ABB RobotStudio station: P2_Main_2.rspag

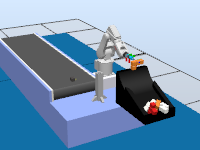
--- station ---
Station P2_Main (saved by RobotStudio 21.1.9385.0)
Controller Controller2, task T_ROB1: task frame (RAPID world) sits at (1547.5, 1227.5, 510) mm in the station
Controller Controller2
  mechanical unit ROB_1: IRB120_3_58__01, 6 joints, base frame (0, 0, 0) mm
Layout (positions relative to the parent item):
  - IRB120_3_58__01 [mechanism, from Robots\IRB120_3_58_G_01.rslib] at (1547.5, 1227.5, 510) mm; joint values [0.0586, 0.4229, 0.2961, 0.0888, -0.7209, -0.0668] (rad or m)
  - MyNewTool [mechanism] at (2003, 1250, 900) mm, rotated rx 0 ry 90 rz 0 deg
      TCP MyNewTool at (0, 0, 0) mm, rotated rx 180 ry 0 rz 180 deg
      links: Čep
  - smc_gripper [mechanism, from Parts\smc_gripper.rslib] at (2003, 1250, 900) mm, rotated rx 0 ry 90 rz 0 deg
  - Conv_belt [part] at (-460, 1030, 390) mm, rotated rx 90 ry 0 rz 0 deg
  - Piece_6_L [part] at (2225, 1200, 885.87) mm, rotated rx 0.75 ry 90 rz 90.75 deg
  - Piece_5_S [part] at (2593.69, 1136.23, 500.91) mm, rotated rx -150.15 ry -50.3 rz 82.94 deg
  - Piece_4_T [part] at (2653.03, 1162.05, 521.4) mm, rotated rx -177.09 ry 74.17 rz -180 deg
  - Piece_2_S [part] at (2730.75, 1281.49, 507.1) mm, rotated rx 90 ry 0 rz -176.34 deg
  - Piece_3_L [part] at (2613.74, 1242.05, 481.96) mm, rotated rx -48.71 ry -65.02 rz -0.13 deg
  - Piece_1_T [part] at (3053.29, 1610.48, 33) mm, rotated rx -95.26 ry 5.23 rz -57.48 deg
  - FLIP [part] at (1915, 935, 785) mm, rotated rx 180 ry 0 rz 90 deg
  - PICKUP [part] at (1493.35, 765, 526.5) mm, rotated rx -90 ry 0 rz -90 deg
  - FlipperStand [part] at (1945, 900, 360) mm, rotated rx 90 ry 0 rz 0 deg
  - Environment_6 [part]
  - DROP [part] at (2100, 1525, 950) mm, rotated rx 0 ry 90 rz -90 deg
  - Positioner_1 [smart component, from Components\Positioner.rslib] at (495, 765, 531.5) mm, rotated rx -90 ry 0 rz 0 deg
      properties: Object=Piece_1_T; Position=[0.5 0.765 0.5315]; Orientation=[-1.5707963267949 0 -1.5707963267949]; Reference=Global; ReferenceObject=(none)
  - Positioner_2 [smart component, from Components\Positioner.rslib] at (2954.8, 1487.14, 42.26) mm, rotated rx -84.7 ry -5.18 rz 122.52 deg
      properties: Object=Piece_2_S; Position=[0.35 0.715 0.5315]; Orientation=[-1.5707963267949 0 1.5707963267949]; Reference=Global; ReferenceObject=(none)
  - Positioner_3 [smart component, from Components\Positioner.rslib] at (2714.8, 1530.98, 507.18) mm, rotated rx 89.95 ry 0.02 rz -86.34 deg
      properties: Object=Piece_3_L; Position=[0.1 0.715 0.5315]; Orientation=[-1.5707963267949 0 0]; Reference=Global; ReferenceObject=(none)
  - Positioner_4 [smart component, from Components\Positioner.rslib] at (2552.24, 1285.06, 88.21) mm, rotated rx -95.3 ry 5.18 rz -57.48 deg
      properties: Object=Piece_4_T; Position=[-0.1 0.765 0.5315]; Orientation=[-1.5707963267949 0 -1.5707963267949]; Reference=Global; ReferenceObject=Piece_4_T
  - Positioner_5 [smart component, from Components\Positioner.rslib] at (-250, 715, 531.5) mm, rotated rx -90 ry 0 rz 90 deg
      properties: Object=Piece_5_S; Position=[-0.25 0.715 0.5315]; Orientation=[-1.5707963267949 0 1.5707963267949]; Reference=Global; ReferenceObject=(none)
  - Positioner_6 [smart component, from Components\Positioner.rslib] at (2676.51, 2129.75, 507.42) mm, rotated rx 89.95 ry 0.02 rz -86.34 deg
      properties: Object=Piece_6_L; Position=[-0.5 0.715 0.5315]; Orientation=[-1.5707963267949 0 0]; Reference=Global; ReferenceObject=(none)
  - Attacher_1_G [smart component, from Components\Attacher.rslib]
      properties: Parent=smc_gripper; Flange=0; Child=Piece_1_T; Mount=false; Offset=[0 0 0]; Orientation=[0 0 0]
  - Attacher_2_G [smart component, from Components\Attacher.rslib]
      properties: Parent=smc_gripper; Flange=0; Child=Piece_2_S; Mount=false; Offset=[0 0 0]; Orientation=[0 0 0]
  - Attacher_3_G [smart component, from Components\Attacher.rslib]
      properties: Parent=smc_gripper; Flange=0; Child=Piece_3_L; Mount=false; Offset=[0 0 0]; Orientation=[0 0 0]
  - Attacher_4_G [smart component, from Components\Attacher.rslib]
      properties: Parent=smc_gripper; Flange=0; Child=Piece_4_T; Mount=false; Offset=[0 0 0]; Orientation=[0 0 0]
  - Attacher_5_G [smart component, from Components\Attacher.rslib]
      properties: Parent=smc_gripper; Flange=0; Child=Piece_5_S; Mount=false; Offset=[0 0 0]; Orientation=[0 0 0]
  - Attacher_6_G [smart component, from Components\Attacher.rslib]
      properties: Parent=smc_gripper; Flange=0; Child=Piece_6_L; Mount=false; Offset=[0 0 0]; Orientation=[0 0 0]
  - Detacher_1 [smart component, from Components\Detacher.rslib]
      properties: Child=Piece_1_T; KeepPosition=true
  - Detacher_2 [smart component, from Components\Detacher.rslib]
      properties: Child=Piece_2_S; KeepPosition=true
  - Detacher_3 [smart component, from Components\Detacher.rslib]
      properties: Child=Piece_3_L; KeepPosition=true
  - Detacher_4 [smart component, from Components\Detacher.rslib]
      properties: Child=Piece_4_T; KeepPosition=true
  - Detacher_5 [smart component, from Components\Detacher.rslib]
      properties: Child=Piece_5_S; KeepPosition=true
  - Detacher_6 [smart component, from Components\Detacher.rslib]
      properties: Child=Piece_6_L; KeepPosition=true
  - Conv_placeholder [part] at (1552.8, 750, 531.5) mm
  - Positioner_7 [smart component, from Components\Positioner.rslib] at (2452.35, 1411.66, 333.91) mm, rotated rx 67.53 ry -33.65 rz -60.36 deg
      properties: Object=Conv_placeholder; Position=[-0.6 0.75 0.5315]; Orientation=[0 0 0]; Reference=Global; ReferenceObject=(none)
  - Attacher_1_C [smart component, from Components\Attacher.rslib]
      properties: Parent=Conv_placeholder; Flange=0; Child=Piece_1_T; Mount=false; Offset=[0 0 0]; Orientation=[0 0 0]
  - Attacher_2_C [smart component, from Components\Attacher.rslib]
      properties: Parent=Conv_placeholder; Flange=0; Child=Piece_2_S; Mount=false; Offset=[0 0 0]; Orientation=[0 0 0]
  - Attacher_3_C [smart component, from Components\Attacher.rslib]
      properties: Parent=Conv_placeholder; Flange=0; Child=Piece_3_L; Mount=false; Offset=[0 0 0]; Orientation=[0 0 0]
  - Attacher_4_C [smart component, from Components\Attacher.rslib]
      properties: Parent=Conv_placeholder; Flange=0; Child=Piece_4_T; Mount=false; Offset=[0 0 0]; Orientation=[0 0 0]
  - Attacher_5_C [smart component, from Components\Attacher.rslib]
      properties: Parent=Conv_placeholder; Flange=0; Child=Piece_5_S; Mount=false; Offset=[0 0 0]; Orientation=[0 0 0]
  - Attacher_6_C [smart component, from Components\Attacher.rslib]
      properties: Parent=Conv_placeholder; Flange=0; Child=Piece_6_L; Mount=false; Offset=[0 0 0]; Orientation=[0 0 0]
  - PlaneSensor [smart component, from Components\PlaneSensor.rslib]
      properties: Origin=[1.575 0.73 0.52]; Axis1=[0 0.065 0]; Axis2=[0 0 0.02]; SensedPart=Conv_placeholder
    - _sensorPart_ [part]
  - LogicGate [smart component, from Components\LogicGate.rslib]
      properties: Operator=NOT; Delay=0
  - LogicGate_2 [smart component, from Components\LogicGate.rslib]
      properties: Operator=AND; Delay=0
  - LinearMover_Conv [smart component, from Components\LinearMover.rslib]
      properties: Object=Conv_placeholder; Direction=[0.005 0 0]; Speed=0.15; Reference=Global; ReferenceObject=(none)
  - LinearMover_1_L [smart component, from Components\LinearMover2.rslib]
      properties: Object=IRB120_3_58__01; Direction=[0 -0.05 0]; Distance=0.05; Duration=1; Reference=Global; ReferenceObject=(none)
  - LinearMover_2_L [smart component, from Components\LinearMover2.rslib]
      properties: Object=Piece_2_S; Direction=[0 -0.05 0]; Distance=0.05; Duration=1; Reference=Global; ReferenceObject=(none)
  - LinearMover_3_L [smart component, from Components\LinearMover2.rslib]
      properties: Object=Piece_3_L; Direction=[0 -0.05 0]; Distance=0.05; Duration=1; Reference=Global; ReferenceObject=(none)
  - LinearMover_4_L [smart component, from Components\LinearMover2.rslib]
      properties: Object=Piece_4_T; Direction=[-0.05 0 0]; Distance=0.05; Duration=1; Reference=Global; ReferenceObject=(none)
  - LinearMover_5_L [smart component, from Components\LinearMover2.rslib]
      properties: Object=Piece_5_S; Direction=[1 0 0]; Distance=0; Duration=0; Reference=Global; ReferenceObject=(none)
  - LinearMover_6_L [smart component, from Components\LinearMover2.rslib]
      properties: Object=Piece_6_L; Direction=[0 -0.05 0]; Distance=0.05; Duration=1; Reference=Global; ReferenceObject=(none)
  - Slide [part] at (2100, 1450, 375) mm, rotated rx 90 ry 0 rz 0 deg
  - Frame_1 [frame] at (0, 0, 60) mm
Attachment: MyNewTool is attached to IRB120_3_58__01 / Link6
Attachment: smc_gripper is attached to IRB120_3_58__01 / Link6
Attachment: Positioner_6 is attached to Piece_2_S
Attachment: Positioner_4 is attached to Piece_1_T
Attachment: Positioner_3 is attached to Piece_2_S
Attachment: Positioner_2 is attached to Piece_1_T
Attachment: Positioner_1 is attached to FlipperStand
Attachment: Positioner_7 is attached to Piece_5_S
Station signals: DI DET_ALL, DI ATT_CONV, DI POS_RESET
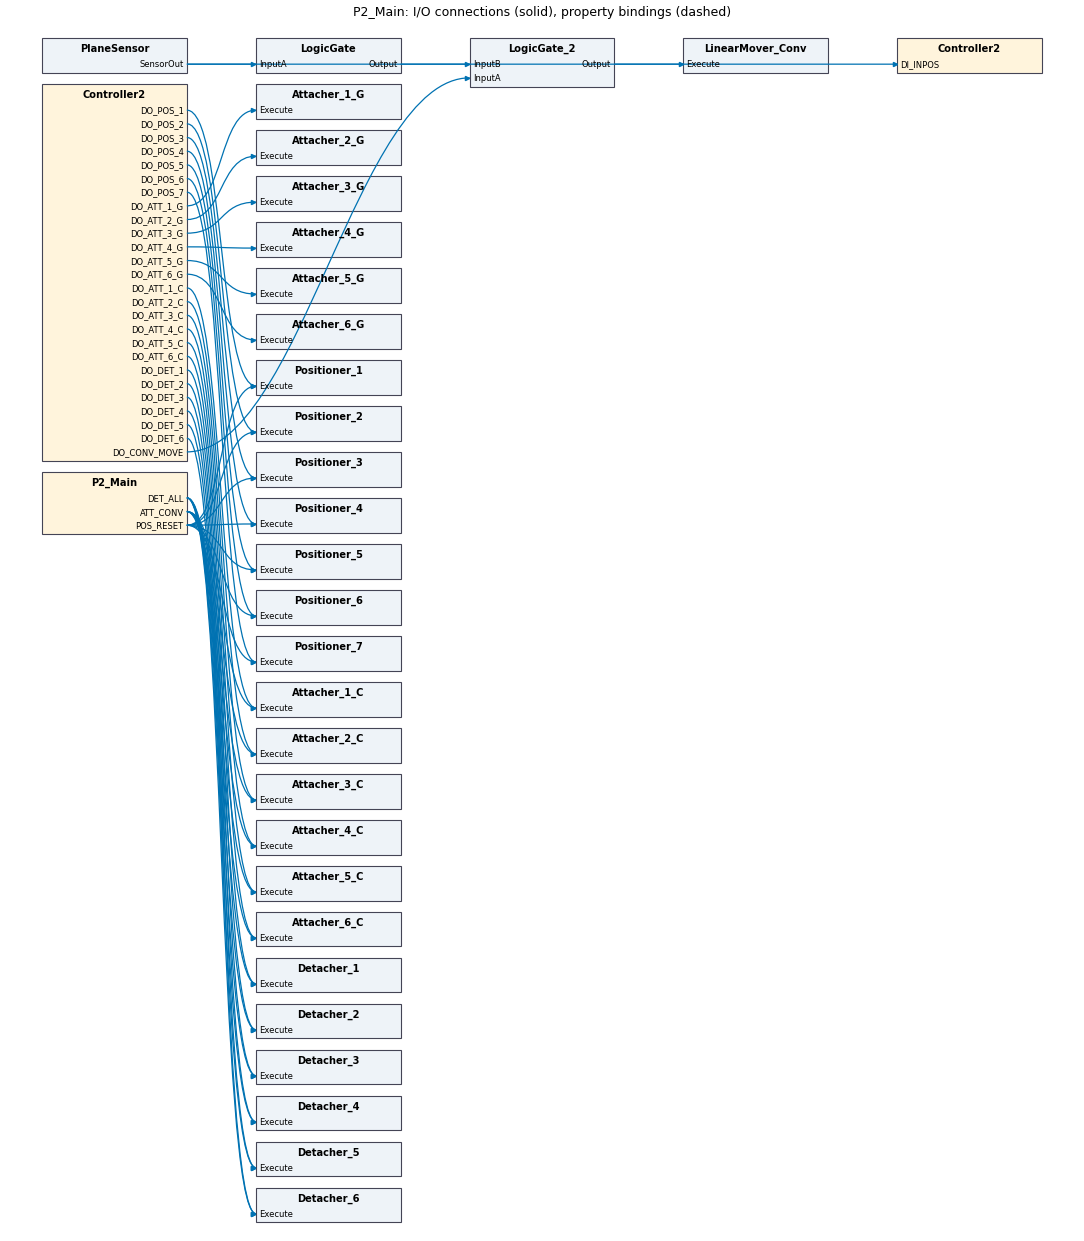
Station logic (signal -> signal, property => property):
  PlaneSensor.SensorOut -> LogicGate.InputA
  LogicGate.Output -> LogicGate_2.InputB
  LogicGate_2.Output -> LinearMover_Conv.Execute
  Controller2.DO_POS_1 -> Positioner_1.Execute
  Controller2.DO_POS_2 -> Positioner_2.Execute
  Controller2.DO_POS_3 -> Positioner_3.Execute
  Controller2.DO_POS_4 -> Positioner_4.Execute
  Controller2.DO_POS_5 -> Positioner_5.Execute
  Controller2.DO_POS_6 -> Positioner_6.Execute
  Controller2.DO_POS_7 -> Positioner_7.Execute
  Controller2.DO_ATT_1_G -> Attacher_1_G.Execute
  Controller2.DO_ATT_2_G -> Attacher_2_G.Execute
  Controller2.DO_ATT_3_G -> Attacher_3_G.Execute
  Controller2.DO_ATT_4_G -> Attacher_4_G.Execute
  Controller2.DO_ATT_5_G -> Attacher_5_G.Execute
  Controller2.DO_ATT_6_G -> Attacher_6_G.Execute
  Controller2.DO_ATT_1_C -> Attacher_1_C.Execute
  Controller2.DO_ATT_2_C -> Attacher_2_C.Execute
  Controller2.DO_ATT_3_C -> Attacher_3_C.Execute
  Controller2.DO_ATT_4_C -> Attacher_4_C.Execute
  Controller2.DO_ATT_5_C -> Attacher_5_C.Execute
  Controller2.DO_ATT_6_C -> Attacher_6_C.Execute
  Controller2.DO_DET_1 -> Detacher_1.Execute
  Controller2.DO_DET_2 -> Detacher_2.Execute
  Controller2.DO_DET_3 -> Detacher_3.Execute
  Controller2.DO_DET_4 -> Detacher_4.Execute
  Controller2.DO_DET_5 -> Detacher_5.Execute
  Controller2.DO_DET_6 -> Detacher_6.Execute
  Controller2.DO_CONV_MOVE -> LogicGate_2.InputA
  PlaneSensor.SensorOut -> Controller2.DI_INPOS
  P2_Main.DET_ALL -> Detacher_1.Execute
  P2_Main.DET_ALL -> Detacher_2.Execute
  P2_Main.DET_ALL -> Detacher_3.Execute
  P2_Main.DET_ALL -> Detacher_4.Execute
  P2_Main.DET_ALL -> Detacher_5.Execute
  P2_Main.DET_ALL -> Detacher_6.Execute
  P2_Main.ATT_CONV -> Attacher_1_C.Execute
  P2_Main.ATT_CONV -> Attacher_2_C.Execute
  P2_Main.ATT_CONV -> Attacher_3_C.Execute
  P2_Main.ATT_CONV -> Attacher_4_C.Execute
  P2_Main.ATT_CONV -> Attacher_5_C.Execute
  P2_Main.ATT_CONV -> Attacher_6_C.Execute
  P2_Main.POS_RESET -> Positioner_1.Execute
  P2_Main.POS_RESET -> Positioner_2.Execute
  P2_Main.POS_RESET -> Positioner_3.Execute
  P2_Main.POS_RESET -> Positioner_5.Execute
  P2_Main.POS_RESET -> Positioner_6.Execute
  P2_Main.POS_RESET -> Positioner_7.Execute
  P2_Main.POS_RESET -> Positioner_4.Execute
Targets, tools, work objects and paths stored in the station and not in the controller backup, written as RAPID:
! task T_ROB1
MODULE Module1
  CONST robtarget P_4:=[[381.789321861,-391.789321901,490],[0.653281482,0.27059805,0.653281482,-0.27059805],[-1,-1,0,1],[9E+09,9E+09,9E+09,9E+09,9E+09,9E+09]];
ENDMODULE


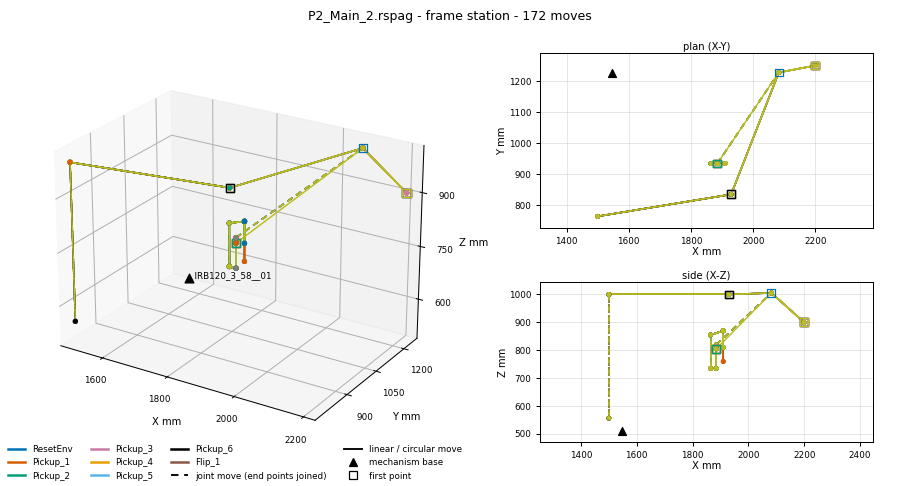
[picture p0: tool path of P2_Main_2.rspag in frame station, 172 of 172 moves have a stored position in this frame; points joined in program order, loops and branches not executed]
--- Backups/Controller2/RAPID/TASK1/PROGMOD/CalibData.mod ---
MODULE CalibData
    PERS tooldata MyNewTool:=[TRUE,[[0,0,60],[1,0,0,0]],[0.3,[0,0,30.653],[1,0,0,0],0,0,0]];
    PERS tooldata smc_gripper:=[TRUE,[[0,0.004,197.001],[1,0,0,0]],[1,[0.207,-0.496,71.18],[1,0,0,0],0,0,0]];
ENDMODULE

--- Backups/Controller2/RAPID/TASK1/PROGMOD/Module1.mod ---
MODULE Module1
    CONST robtarget P_1:=[[381.789321861,-391.789321901,490],[0.653281482,0.27059805,0.653281482,-0.27059805],[-1,-1,0,1],[9E+09,9E+09,9E+09,9E+09,9E+09,9E+09]];
    CONST robtarget P_2:=[[-47.5,-462.5,490],[0,0,-0.707106781,0.707106781],[-2,-1,-1,1],[9E+09,9E+09,9E+09,9E+09,9E+09,9E+09]];
    CONST robtarget P_3:=[[-47.5,-462.5,46.5],[0,0,1,0],[-2,0,2,0],[9E+09,9E+09,9E+09,9E+09,9E+09,9E+09]];

    CONST robtarget D:=[[652.5,22.5,390],[0.707106781,0,0.707106781,0],[0,0,-1,1],[9E+09,9E+09,9E+09,9E+09,9E+09,9E+09]];
    CONST robtarget Standby_1:=[[534.962,0.004,495.5],[0.707106781,0,0.707106781,0],[0,-1,0,1],[9E+09,9E+09,9E+09,9E+09,9E+09,9E+09]];

    CONST robtarget F_1:=[[337.5,-292.5,295],[0.5,-0.5,0.5,-0.5],[-1,1,-3,0],[9E+09,9E+09,9E+09,9E+09,9E+09,9E+09]];
    CONST robtarget F_1R:=[[337.5,-292.5,310],[0.707106781,0,0.707106781,0],[-1,1,-2,0],[9E+09,9E+09,9E+09,9E+09,9E+09,9E+09]];
    CONST robtarget F_2:=[[337.5,-292.5,225],[0.5,-0.5,0.5,-0.5],[-1,1,-3,0],[9E+09,9E+09,9E+09,9E+09,9E+09,9E+09]];
    CONST robtarget F_3:=[[317.5,-292.5,225],[0.5,-0.5,0.5,-0.5],[-1,1,-3,0],[9E+09,9E+09,9E+09,9E+09,9E+09,9E+09]];
    CONST robtarget F_4:=[[317.5,-292.5,345],[0,0,1,0],[-1,0,-1,0],[9E+09,9E+09,9E+09,9E+09,9E+09,9E+09]];
    CONST robtarget F_5:=[[362.5,-292.5,360],[0,0,1,0],[-1,0,-1,0],[9E+09,9E+09,9E+09,9E+09,9E+09,9E+09]];
    CONST robtarget F_6:=[[362.5,-292.5,300],[0,0,1,0],[-1,0,-1,0],[9E+09,9E+09,9E+09,9E+09,9E+09,9E+09]];
    CONST robtarget F_5R:=[[362.5,-292.5,360],[0,1,0,0],[-1,0,1,0],[9E+09,9E+09,9E+09,9E+09,9E+09,9E+09]];
    CONST robtarget F_6R:=[[362.5,-292.5,300],[0,1,0,0],[-1,0,1,0],[9E+09,9E+09,9E+09,9E+09,9E+09,9E+09]];

    VAR num CASE_NO := 0;



    PROC main()

        TEST CASE_NO
            CASE 0:
                ResetEnv;
                Start;

                CASE_NO := 1;

            CASE 1:
                WaitDI DI_INPOS, 1;
                Pickup_1;
                Flip_1;

                WaitTime 2;
                Drop_1;

                CASE_NO := 2;

            CASE 2:
                Pickup_2;
                Flip_2;
                WaitTime 2;
                Drop_2;

                CASE_NO := 3;

            CASE 3:
                Pickup_3;
                Flip_3;
                WaitTime 2;
                Drop_3;

                CASE_NO := 4;

            CASE 4:
                Pickup_4;
                Flip_4;
                WaitTime 2;
                Drop_4;

                CASE_NO := 5;

            CASE 5:
                Pickup_5;
                Flip_5;
                WaitTime 2;
                Drop_5;

                CASE_NO := 6;

            CASE 6:
                Pickup_6;
                Flip_6;
                WaitTime 2;
                Drop_6;

                CASE_NO := 7;

            CASE 7:


                CASE_NO := 8;

            CASE 8:


                CASE_NO := 9;

            CASE 9:


                CASE_NO := 10;

            CASE 10:


                CASE_NO := 11;

            CASE 11:


                CASE_NO := 12;

            CASE 12:


                CASE_NO := 13;

            CASE 13:

                Break;

        ENDTEST

    ENDPROC

    PROC ResetEnv()
        SetDO DO_CONV_MOVE, 0;

        PulseDO DO_DET_1;
        PulseDO DO_DET_2;
        PulseDO DO_DET_3;
        PulseDO DO_DET_4;
        PulseDO DO_DET_5;
        PulseDO DO_DET_6;

        PulseDO DO_POS_1;
        PulseDO DO_POS_2;
        PulseDO DO_POS_3;
        PulseDO DO_POS_4;
        PulseDO DO_POS_5;
        PulseDO DO_POS_6;
        PulseDO DO_POS_7;

        MoveL Standby_1,v100,fine,smc_gripper\WObj:=wobj0;

    ENDPROC

    PROC Start()
        PulseDO DO_ATT_1_C;
        PulseDO DO_ATT_2_C;
        PulseDO DO_ATT_3_C;
        PulseDO DO_ATT_4_C;
        PulseDO DO_ATT_5_C;
        PulseDO DO_ATT_6_C;

        SetDO DO_CONV_MOVE, 1;
        WaitDI DI_INPOS, 1;
    ENDPROC

    PROC Pickup_1()
        MoveL P_1,v1000,fine,smc_gripper\WObj:=wobj0;
        MoveL P_2,v1000,fine,smc_gripper\WObj:=wobj0;
        MoveJ P_3,v1000,fine,smc_gripper\WObj:=wobj0;
        PulseDO DO_DET_1;
        WaitTime 0.25;
        PulseDO DO_ATT_1_G;
        MoveJ P_2,v1000,z200,smc_gripper\WObj:=wobj0;
        MoveL P_1,v1000,fine,smc_gripper\WObj:=wobj0;
        MoveL Standby_1,v1000,fine,smc_gripper\WObj:=wobj0;
    ENDPROC

    PROC Pickup_2()
        MoveL P_1,v1000,fine,smc_gripper\WObj:=wobj0;
        MoveL P_2,v1000,fine,smc_gripper\WObj:=wobj0;
        MoveJ P_3,v1000,fine,smc_gripper\WObj:=wobj0;
        PulseDO DO_DET_2;
        WaitTime 0.25;
        PulseDO DO_ATT_2_G;
        MoveJ P_2,v1000,z200,smc_gripper\WObj:=wobj0;
        MoveL P_1,v1000,fine,smc_gripper\WObj:=wobj0;
        MoveL Standby_1,v1000,fine,smc_gripper\WObj:=wobj0;
    ENDPROC

    PROC Pickup_3()
        MoveL P_1,v1000,fine,smc_gripper\WObj:=wobj0;
        MoveL P_2,v1000,fine,smc_gripper\WObj:=wobj0;
        MoveJ P_3,v1000,fine,smc_gripper\WObj:=wobj0;
        PulseDO DO_DET_3;
        WaitTime 0.25;
        PulseDO DO_ATT_3_G;
        MoveJ P_2,v1000,z200,smc_gripper\WObj:=wobj0;
        MoveL P_1,v1000,fine,smc_gripper\WObj:=wobj0;
        MoveL Standby_1,v1000,fine,smc_gripper\WObj:=wobj0;
    ENDPROC

    PROC Pickup_4()
        MoveL P_1,v1000,fine,smc_gripper\WObj:=wobj0;
        MoveL P_2,v1000,fine,smc_gripper\WObj:=wobj0;
        MoveJ P_3,v1000,fine,smc_gripper\WObj:=wobj0;
        PulseDO DO_DET_4;
        WaitTime 0.25;
        PulseDO DO_ATT_4_G;
        MoveJ P_2,v1000,z200,smc_gripper\WObj:=wobj0;
        MoveL P_1,v1000,fine,smc_gripper\WObj:=wobj0;
        MoveL Standby_1,v1000,fine,smc_gripper\WObj:=wobj0;
    ENDPROC

    PROC Pickup_5()
        MoveL P_1,v1000,fine,smc_gripper\WObj:=wobj0;
        MoveL P_2,v1000,fine,smc_gripper\WObj:=wobj0;
        MoveJ P_3,v1000,fine,smc_gripper\WObj:=wobj0;
        PulseDO DO_DET_5;
        WaitTime 0.25;
        PulseDO DO_ATT_5_G;
        MoveJ P_2,v1000,z200,smc_gripper\WObj:=wobj0;
        MoveL P_1,v1000,fine,smc_gripper\WObj:=wobj0;
        MoveL Standby_1,v1000,fine,smc_gripper\WObj:=wobj0;
    ENDPROC

    PROC Pickup_6()
        MoveL P_1,v1000,fine,smc_gripper\WObj:=wobj0;
        MoveL P_2,v1000,fine,smc_gripper\WObj:=wobj0;
        MoveJ P_3,v1000,fine,smc_gripper\WObj:=wobj0;
        PulseDO DO_DET_6;
        WaitTime 0.25;
        PulseDO DO_ATT_6_G;
        MoveJ P_2,v1000,z200,smc_gripper\WObj:=wobj0;
        MoveL P_1,v1000,fine,smc_gripper\WObj:=wobj0;
        MoveL Standby_1,v1000,fine,smc_gripper\WObj:=wobj0;
    ENDPROC

    PROC Flip_1()
        MoveJ F_1,v1000,fine,smc_gripper\WObj:=wobj0;
        MoveL F_2,v1000,fine,smc_gripper\WObj:=wobj0;
        PulseDO DO_DET_1;
        WaitTime 0.25;
        MoveL F_3,v1000,z100,smc_gripper\WObj:=wobj0;
        MoveL F_4,v1000,z100,smc_gripper\WObj:=wobj0;
        MoveL F_5,v1000,z100,smc_gripper\WObj:=wobj0;
        MoveL F_6,v1000,fine,smc_gripper\WObj:=wobj0;
        PulseDO DO_ATT_1_G;
        WaitTime 0.25;
        MoveL F_5,v1000,z100,smc_gripper\WObj:=wobj0;
        MoveL F_5R,v1000,z100,smc_gripper\WObj:=wobj0;
        MoveL F_6R,v1000,fine,smc_gripper\WObj:=wobj0;
        PulseDO DO_DET_1;
        WaitTime 0.25;
        MoveL F_5,v1000,z100,smc_gripper\WObj:=wobj0;
        MoveL F_4,v1000,z100,smc_gripper\WObj:=wobj0;
        MoveL F_3,v1000,z100,smc_gripper\WObj:=wobj0;
        MoveL F_2,v1000,fine,smc_gripper\WObj:=wobj0;
        PulseDO DO_ATT_1_G;
        WaitTime 0.25;
        MoveL F_1,v1000,z100,smc_gripper\WObj:=wobj0;
        MoveL F_1R,v1000,z100,smc_gripper\WObj:=wobj0;
        MoveJ Standby_1,v1000,fine,smc_gripper\WObj:=wobj0;
    ENDPROC

    PROC Flip_2()
        MoveJ F_1,v1000,fine,smc_gripper\WObj:=wobj0;
        MoveL F_2,v1000,fine,smc_gripper\WObj:=wobj0;
        PulseDO DO_DET_2;
        WaitTime 0.25;
        MoveL F_3,v1000,z100,smc_gripper\WObj:=wobj0;
        MoveL F_4,v1000,z100,smc_gripper\WObj:=wobj0;
        MoveL F_5,v1000,z100,smc_gripper\WObj:=wobj0;
        MoveL Offs(F_6, 0, 0, -50), v1000, fine, smc_gripper\WObj:=wobj0;
        PulseDO DO_ATT_2_G;
        WaitTime 0.25;
        MoveL F_5,v1000,z100,smc_gripper\WObj:=wobj0;
        MoveL F_5R,v1000,z100,smc_gripper\WObj:=wobj0;
        MoveL Offs(F_6R, 0, 0, -50), v1000, fine, smc_gripper\WObj:=wobj0;
        PulseDO DO_DET_2;
        WaitTime 0.25;
        MoveL F_5,v1000,z100,smc_gripper\WObj:=wobj0;
        MoveL F_4,v1000,z100,smc_gripper\WObj:=wobj0;
        MoveL F_3,v1000,z100,smc_gripper\WObj:=wobj0;
        MoveL F_2,v1000,fine,smc_gripper\WObj:=wobj0;
        PulseDO DO_ATT_2_G;
        WaitTime 0.25;
        MoveL F_1,v1000,z100,smc_gripper\WObj:=wobj0;
        MoveL F_1R,v1000,z100,smc_gripper\WObj:=wobj0;
        MoveJ Standby_1,v1000,fine,smc_gripper\WObj:=wobj0;
    ENDPROC

    PROC Flip_3()
        MoveJ F_1,v1000,fine,smc_gripper\WObj:=wobj0;
        MoveL F_2,v1000,fine,smc_gripper\WObj:=wobj0;
        PulseDO DO_DET_3;
        WaitTime 0.25;
        MoveL F_3,v1000,z100,smc_gripper\WObj:=wobj0;
        MoveL F_4,v1000,z100,smc_gripper\WObj:=wobj0;
        MoveL F_5,v1000,z100,smc_gripper\WObj:=wobj0;
        MoveL F_6,v1000,fine,smc_gripper\WObj:=wobj0;
        PulseDO DO_ATT_3_G;
        WaitTime 0.25;
        MoveL F_5,v1000,z100,smc_gripper\WObj:=wobj0;
        MoveL F_5R,v1000,z100,smc_gripper\WObj:=wobj0;
        MoveL F_6R,v1000,fine,smc_gripper\WObj:=wobj0;
        PulseDO DO_DET_3;
        WaitTime 0.25;
        MoveL F_5,v1000,z100,smc_gripper\WObj:=wobj0;
        MoveL F_4,v1000,z100,smc_gripper\WObj:=wobj0;
        MoveL F_3,v1000,z100,smc_gripper\WObj:=wobj0;
        MoveL F_2,v1000,fine,smc_gripper\WObj:=wobj0;
        PulseDO DO_ATT_3_G;
        WaitTime 0.25;
        MoveL F_1,v1000,z100,smc_gripper\WObj:=wobj0;
        MoveL F_1R,v1000,z100,smc_gripper\WObj:=wobj0;
        MoveJ Standby_1,v1000,fine,smc_gripper\WObj:=wobj0;
    ENDPROC

    PROC Flip_4()
        MoveJ F_1,v1000,fine,smc_gripper\WObj:=wobj0;
        MoveL F_2,v1000,fine,smc_gripper\WObj:=wobj0;
        PulseDO DO_DET_4;
        WaitTime 0.25;
        MoveL F_3,v1000,z100,smc_gripper\WObj:=wobj0;
        MoveL F_4,v1000,z100,smc_gripper\WObj:=wobj0;
        MoveL F_5,v1000,z100,smc_gripper\WObj:=wobj0;
        MoveL F_6,v1000,fine,smc_gripper\WObj:=wobj0;
        PulseDO DO_ATT_4_G;
        WaitTime 0.25;
        MoveL F_5,v1000,z100,smc_gripper\WObj:=wobj0;
        MoveL F_5R,v1000,z100,smc_gripper\WObj:=wobj0;
        MoveL F_6R,v1000,fine,smc_gripper\WObj:=wobj0;
        PulseDO DO_DET_4;
        WaitTime 0.25;
        MoveL F_5,v1000,z100,smc_gripper\WObj:=wobj0;
        MoveL F_4,v1000,z100,smc_gripper\WObj:=wobj0;
        MoveL F_3,v1000,z100,smc_gripper\WObj:=wobj0;
        MoveL F_2,v1000,fine,smc_gripper\WObj:=wobj0;
        PulseDO DO_ATT_4_G;
        WaitTime 0.25;
        MoveL F_1,v1000,z100,smc_gripper\WObj:=wobj0;
        MoveL F_1R,v1000,z100,smc_gripper\WObj:=wobj0;
        MoveJ Standby_1,v1000,fine,smc_gripper\WObj:=wobj0;
    ENDPROC

    PROC Flip_5()
        MoveJ F_1,v1000,fine,smc_gripper\WObj:=wobj0;
        MoveL F_2,v1000,fine,smc_gripper\WObj:=wobj0;
        PulseDO DO_DET_5;
        WaitTime 0.25;
        MoveL F_3,v1000,z100,smc_gripper\WObj:=wobj0;
        MoveL F_4,v1000,z100,smc_gripper\WObj:=wobj0;
        MoveL F_5,v1000,z100,smc_gripper\WObj:=wobj0;
        MoveL Offs(F_6, 0, 0, -50), v1000, fine, smc_gripper\WObj:=wobj0;
        PulseDO DO_ATT_5_G;
        WaitTime 0.25;
        MoveL F_5,v1000,z100,smc_gripper\WObj:=wobj0;
        MoveL F_5R,v1000,z100,smc_gripper\WObj:=wobj0;
        MoveL Offs(F_6R, 0, 0, -50), v1000, fine, smc_gripper\WObj:=wobj0;
        PulseDO DO_DET_5;
        WaitTime 0.25;
        MoveL F_5,v1000,z100,smc_gripper\WObj:=wobj0;
        MoveL F_4,v1000,z100,smc_gripper\WObj:=wobj0;
        MoveL F_3,v1000,z100,smc_gripper\WObj:=wobj0;
        MoveL F_2,v1000,fine,smc_gripper\WObj:=wobj0;
        PulseDO DO_ATT_5_G;
        WaitTime 0.25;
        MoveL F_1,v1000,z100,smc_gripper\WObj:=wobj0;
        MoveL F_1R,v1000,z100,smc_gripper\WObj:=wobj0;
        MoveJ Standby_1,v1000,fine,smc_gripper\WObj:=wobj0;
    ENDPROC

    PROC Flip_6()
        MoveJ F_1,v1000,fine,smc_gripper\WObj:=wobj0;
        MoveL F_2,v1000,fine,smc_gripper\WObj:=wobj0;
        PulseDO DO_DET_6;
        WaitTime 0.25;
        MoveL F_3,v1000,z100,smc_gripper\WObj:=wobj0;
        MoveL F_4,v1000,z100,smc_gripper\WObj:=wobj0;
        MoveL F_5,v1000,z100,smc_gripper\WObj:=wobj0;
        MoveL F_6,v1000,fine,smc_gripper\WObj:=wobj0;
        PulseDO DO_ATT_6_G;
        WaitTime 0.25;
        MoveL F_5,v1000,z100,smc_gripper\WObj:=wobj0;
        MoveL F_5R,v1000,z100,smc_gripper\WObj:=wobj0;
        MoveL F_6R,v1000,fine,smc_gripper\WObj:=wobj0;
        PulseDO DO_DET_6;
        WaitTime 0.25;
        MoveL F_5,v1000,z100,smc_gripper\WObj:=wobj0;
        MoveL F_4,v1000,z100,smc_gripper\WObj:=wobj0;
        MoveL F_3,v1000,z100,smc_gripper\WObj:=wobj0;
        MoveL F_2,v1000,fine,smc_gripper\WObj:=wobj0;
        PulseDO DO_ATT_6_G;
        WaitTime 0.25;
        MoveL F_1,v1000,z100,smc_gripper\WObj:=wobj0;
        MoveL F_1R,v1000,z100,smc_gripper\WObj:=wobj0;
        MoveJ Standby_1,v1000,fine,smc_gripper\WObj:=wobj0;
    ENDPROC

    PROC Drop_1()
        MoveL D,v1000,z100,smc_gripper\WObj:=wobj0;
        WaitTime 0.25;
        PulseDO DO_DET_1;
        MoveL Standby_1,v1000,z100,smc_gripper\WObj:=wobj0;
    ENDPROC

    PROC Drop_2()
        MoveL D,v1000,fine,smc_gripper\WObj:=wobj0;
        WaitTime 0.25;
        PulseDO DO_DET_2;
        MoveL Standby_1,v1000,z100,smc_gripper\WObj:=wobj0;
    ENDPROC

    PROC Drop_3()
        MoveL D,v1000,fine,smc_gripper\WObj:=wobj0;
        WaitTime 0.25;
        PulseDO DO_DET_3;
        MoveL Standby_1,v1000,z100,smc_gripper\WObj:=wobj0;
    ENDPROC

    PROC Drop_4()
        MoveL D,v1000,fine,smc_gripper\WObj:=wobj0;
        WaitTime 0.25;
        PulseDO DO_DET_4;
        MoveL Standby_1,v1000,z100,smc_gripper\WObj:=wobj0;
    ENDPROC

    PROC Drop_5()
        MoveL D,v1000,fine,smc_gripper\WObj:=wobj0;
        WaitTime 0.25;
        PulseDO DO_DET_5;
        MoveL Standby_1,v1000,z100,smc_gripper\WObj:=wobj0;
    ENDPROC

    PROC Drop_6()
        MoveL D,v1000,fine,smc_gripper\WObj:=wobj0;
        WaitTime 0.25;
        PulseDO DO_DET_6;
        MoveL Standby_1,v1000,z100,smc_gripper\WObj:=wobj0;
    ENDPROC
    PROC TestPath()
        MoveL D,v1000,z100,smc_gripper\WObj:=wobj0;
        MoveL Standby_1,v1000,z100,smc_gripper\WObj:=wobj0;
        MoveL P_1,v1000,z100,smc_gripper\WObj:=wobj0;
        MoveL P_2,v1000,z100,smc_gripper\WObj:=wobj0;
        MoveJ P_3,v1000,z100,smc_gripper\WObj:=wobj0;
        MoveJ P_2,v1000,z100,smc_gripper\WObj:=wobj0;
        MoveL P_1,v1000,z100,smc_gripper\WObj:=wobj0;
        MoveL Standby_1,v1000,z100,smc_gripper\WObj:=wobj0;
        MoveL F_1,v1000,z100,smc_gripper\WObj:=wobj0;
        MoveL F_2,v1000,z100,smc_gripper\WObj:=wobj0;
        MoveL F_3,v1000,z100,smc_gripper\WObj:=wobj0;
        MoveJ F_4,v1000,z100,smc_gripper\WObj:=wobj0;
        MoveL F_5,v1000,z100,smc_gripper\WObj:=wobj0;
        MoveL F_6,v1000,z100,smc_gripper\WObj:=wobj0;
        MoveL F_5,v1000,z100,smc_gripper\WObj:=wobj0;
        MoveL F_5R,v1000,z100,smc_gripper\WObj:=wobj0;
        MoveL F_6R,v1000,z100,smc_gripper\WObj:=wobj0;
        MoveL F_5,v1000,z100,smc_gripper\WObj:=wobj0;
        MoveL F_4,v1000,z100,smc_gripper\WObj:=wobj0;
        MoveL F_3,v1000,z100,smc_gripper\WObj:=wobj0;
        MoveL F_2,v1000,z100,smc_gripper\WObj:=wobj0;
        MoveL F_1,v1000,z100,smc_gripper\WObj:=wobj0;
        MoveL F_1R,v1000,z100,smc_gripper\WObj:=wobj0;
        MoveJ Standby_1,v1000,z100,smc_gripper\WObj:=wobj0;
        MoveL D,v1000,z100,smc_gripper\WObj:=wobj0;
        MoveL Standby_1,v1000,z100,smc_gripper\WObj:=wobj0;
        MoveL D,v1000,z100,smc_gripper\WObj:=wobj0;
    ENDPROC

ENDMODULE

--- Backups/Controller2/RAPID/TASK1/PROGMOD/RsTempModule.mod ---
MODULE RsTempModule
    PROC RsTempPath()

    ENDPROC
ENDMODULE

--- Backups/Controller2/SYSPAR/EIO.cfg ---
EIO:CFG_1.0:6:1::
#
EIO_SIGNAL:

      -Name "DO_ATT_1_C" -SignalType "DO"

      -Name "DO_POS_1" -SignalType "DO"

      -Name "DO_POS_2" -SignalType "DO"

      -Name "DO_POS_3" -SignalType "DO"

      -Name "DO_POS_4" -SignalType "DO"

      -Name "DO_POS_5" -SignalType "DO"

      -Name "DO_POS_6" -SignalType "DO"

      -Name "DO_POS_7" -SignalType "DO"

      -Name "DO_ATT_1_G" -SignalType "DO"

      -Name "DO_ATT_2_G" -SignalType "DO"

      -Name "DO_ATT_3_G" -SignalType "DO"

      -Name "DO_ATT_4_G" -SignalType "DO"

      -Name "DO_ATT_5_G" -SignalType "DO"

      -Name "DO_ATT_6_G" -SignalType "DO"

      -Name "DO_ATT_2_C" -SignalType "DO"

      -Name "DO_ATT_3_C" -SignalType "DO"

      -Name "DO_ATT_4_C" -SignalType "DO"

      -Name "DO_ATT_5_C" -SignalType "DO"

      -Name "DO_ATT_6_C" -SignalType "DO"

      -Name "DO_DET_1" -SignalType "DO"

      -Name "DO_DET_2" -SignalType "DO"

      -Name "DO_DET_3" -SignalType "DO"

      -Name "DO_DET_4" -SignalType "DO"

      -Name "DO_DET_5" -SignalType "DO"

      -Name "DO_DET_6" -SignalType "DO"

      -Name "DO_CONV_MOVE" -SignalType "DO"

      -Name "DI_INPOS" -SignalType "DI"
